// TIA Portal V21 export
TYPE "coneCrusherSimCmd"
   STRUCT
      simEn : Bool;
      invertPrestartAlm : Bool;
      oilPump1Fault : Bool;
      oilPump2Fault : Bool;
      premolding : Bool;
   END_STRUCT;
END_TYPE
